Universal Robots PolyScope program: RuchP1MS.urp

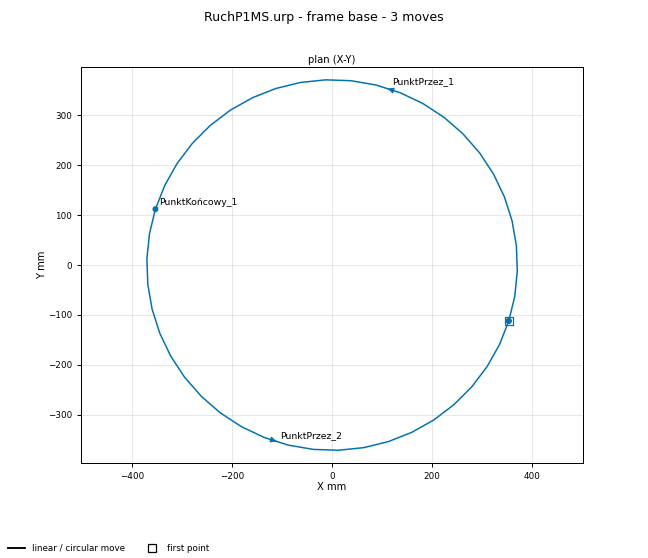
[picture p0: tool path of RuchP1MS.urp in frame base, 3 of 5 moves have a stored position in this frame; points joined in program order, loops and branches not executed]
Program RuchP1MS (installation=default directory=/programs/usbdisk createdIn=3.15.8.106339 lastSavedIn=3.15.8.106339 robotSerialNumber=2020330428)
Calibrated DH parameters: a=[0.000029, -0.241913, -0.128453, -0.000049, -0.000012, 0]; d=[0.151842, -4.082088, 33.504745, -29.309875, 0.08529, 0.082285]; alpha=[1.571059, -0.006644, 0.005794, 1.571984, -1.571997, 0]; deltaTheta=[-0.000032, 0.111537, 0.813391, -0.924919, 0.000036, 0.000016]
Robot Program (runOnlyOnce=false)
  MoveP speed 200 mm/s, acceleration 1200 mm/s^2 (blendRadius=0.001 useActiveTCP=true) feature=Base
    Waypoint Punkt_orienta_1: motionParameters(blendRadius=0); TCP in base x=353.728 y=-111.92 z=116.893 mm, rx=2.2251 ry=-2.2131 rz=0.0025 rad; joints [0.003, -110.002, -99.999, -60, 90.002, 0] deg; flange x=353.817 y=-111.662 z=191.892 mm, rx=2.2251 ry=-2.2131 rz=0.0025 rad
    CircleMove (OrientationMode=FIXED)
      Waypoint PunktPrzez_1: TCP in base x=111.942 y=353.72 z=116.904 mm, rx=3.1404 ry=0.0084 rz=0.0055 rad; joints [90, -110, -100, -60, 90, 0] deg; flange x=111.682 y=353.808 z=191.903 mm, rx=3.1404 ry=0.0084 rz=0.0055 rad
      Waypoint PunktKońcowy_1: TCP in base x=-353.72 y=111.931 z=116.903 mm, rx=-2.2144 ry=-2.2262 rz=-0.0051 rad; joints [180, -110, -100, -60, 90.004, 0] deg; flange x=-353.808 y=111.676 z=191.903 mm, rx=-2.2144 ry=-2.2262 rz=-0.0051 rad
    CircleMove (OrientationMode=FIXED)
      Waypoint PunktPrzez_2: TCP in base x=-111.948 y=-353.72 z=116.904 mm, rx=0.0084 ry=-3.1381 rz=-0.0018 rad; joints [270, -110, -100, -60, 89.998, 0] deg; flange x=-111.685 y=-353.808 z=191.903 mm, rx=0.0084 ry=-3.1381 rz=-0.0018 rad
      Waypoint PunktKońcowy_2: TCP in base x=353.72 y=-111.95 z=116.904 mm, rx=2.225 ry=-2.2132 rz=0.0026 rad; joints [360, -110, -100, -60, 89.997, 0] deg; flange x=353.808 y=-111.686 z=191.903 mm, rx=2.225 ry=-2.2132 rz=0.0026 rad
    Halt
